TYPE ST_StaRequest :
STRUCT
    AutoInitiate        : BIT; // 
    AutoConfirm         : BIT; // 
    FaultReset          : BIT; // 
    Hold                : BIT; // 
    LampTest            : BIT; // 
    PauseMSG            : BIT; // 
    DryCycle            : BIT; // 
    AllProcessOn        : BIT; // 
    AllProcessOff       : BIT; // 
    ProdCountReset      : BIT; //   
END_STRUCT
END_TYPE

(* stored: Version 1.1.0.1, ProductVersion 3.1.4024.12
   DUT ST_StaRequest: Id {7104d51e-bfde-4984-b2fb-ca98e62e8cda} *)
